TYPE ST_P_GET_RECIPE :
STRUCT
	Barcode:				INT;
	ByCustomField:			BOOL;
	CustomFiled:			STRING;
	Contains:				STRING;
END_STRUCT
END_TYPE

(* stored: Version 1.1.0.1, ProductVersion 3.1.4024.10
   DUT ST_P_GET_RECIPE: Id {1349cb4b-a553-4d89-9e18-40e5b7ef8a72} *)
